KUKA KRL program: chk_w4_wechs_ok.src

&ACCESS RVO9
&REL 1
&COMMENT GUN C3
DEF chk_w4_wechs_ok( )

; VERIFICAÇÃO DE FERRAMENTA: C3

$TIMER[10] = 0
$TIMER_STOP[10] = FALSE

wait for ((($IN[585]) or (not($in[585]) and $in[3320])) and ($in[577] or (not ($IN[577]) and $in[3320])) and ($in[161]) and ($in[177]) and (NOT $in[201]) and ($in[209]) and ($IN[169]) and ($in[185]) AND ($in[219]))

$TIMER_STOP[10] = TRUE
$TIMER[10] = 0

;//---- End -------
;Diag_Appl(#Off,5)

END
